INTERFACE I_ANY EXTENDS I_Datatype

METHOD PUBLIC CanBecome : BOOL
VAR_INPUT
	Target : I_Datatype;
END_VAR
END_METHOD

METHOD PUBLIC Clear
VAR_INPUT
END_VAR
END_METHOD

PROPERTY PUBLIC IsResolved : BOOL
GET
END_GET
END_PROPERTY

METHOD PUBLIC TryBecome : BOOL
VAR_INPUT
	Target : I_Datatype;
END_VAR
END_METHOD

END_INTERFACE

(* stored: Version 1.1.0.1, ProductVersion 3.1.4026.18
   Itf I_ANY: Id {8527ab3c-0e0b-05b3-26dc-9d94eae3bd2a}
   Method CanBecome: Id {724d82c3-b9d4-0fc3-3df0-30f4deb951ea}
   Method Clear: Id {269c7724-ce6a-0b38-0413-25b2ac71b9e4}
   Property IsResolved: Id {e2c5de62-d370-07e4-12cb-3481ef8a3bd1}
   Get Get: Id {bc530904-3701-0093-0c8a-b317ff19d363}
   Method TryBecome: Id {b66fb347-1bad-0ceb-1851-fc2726f42cd7} *)
